PROGRAM MAIN
VAR
	//rTrig : R_TRIG;
	dwTmp : DWORD;
END_VAR

P_InitOnce(); // NBT-NEU 

P_GetTime(); // NBT-NEU 

P_RestoreCurrentLanguage(); // NBT-NEU 

P_InputHandling(); // NBT-NEU 

P_TpKommunikation(); //ehem. FC4 -- OK

P_Betriebsarten(); //ehem. FC2 -- OK

P_Ablauf(); //ehem. FC20 -- OK -- 500er ID-Bereich

P_Sortierer(); //ehem. FC24 -- OK

P_FehlerAllgemein(); //ehem. FC3 -- OK -- 600er ID-Bereich

P_StatusAnzeige(); //ehem. FC95

//P_LetzterFC(); //ehem. FC99

P_OutputHandling(); // OK

P_HmiHandling(); //NBT-NEU

METHOD M_Log : DINT
VAR_INPUT
	reqLevel : WORD; (* 0-Nothing, 1-ErrOnly, 2-Warnings, 4-Info , 8-Verbose *)
	objectName : STRING(40);
	sMsg	: T_MaxString;(* Message string *)
	errNo : UDINT := 16#FFFFFFFF;
END_VAR
VAR
	sTmp : STRING;
END_VAR
IF WORD_TO_BOOL(RVL.currLogLevel AND reqLevel) = TRUE THEN
	
	sTmp := '[';
	sTmp := CONCAT( sTmp, objectName);
	sTmp := CONCAT( sTmp, '], ');
	
	CASE reqLevel OF
	 1:  sTmp := CONCAT( sTmp,'[E] ');
	 2:  sTmp := CONCAT( sTmp,'[W] ');
	 4:  sTmp := CONCAT( sTmp,'[I] ');
	 8:  sTmp := CONCAT( sTmp,'[T] ');
	ELSE 
		sTmp := CONCAT( sTmp,'[...] ');
	END_CASE 

	IF errNo <> 16#FFFFFFFF THEN
		sMsg := CONCAT( sMsg,': ');
		sMsg := CONCAT( sMsg, UDINT_TO_STRING(errNo));
	END_IF
	(*
	{IF defined (LOG_VIA_TCP)}
		LOG_PUSH_MSG(msg := CONCAT( sTmp, sMsg));
	{END_IF}
	*)
	M_Log := ADSLOGSTR( ADSLOG_MSGTYPE_HINT OR ADSLOG_MSGTYPE_LOG, CONCAT( sTmp, '%s' ), sMsg );
END_IF
END_METHOD

END_PROGRAM

(* stored: Version 1.1.0.1, ProductVersion 3.1.4024.3
   POU MAIN: Id {3e924d03-094f-4f3e-9add-d5e64d32ee14}, SpecialFunc None
   Method M_Log: Id {83d80e76-90e5-41a8-a3c5-944026f261b4} *)
